TYPE Cnv_Errors_DUT :
STRUCT
	Error_Word_1:	UINT;
	Error_Word_2:	UINT;
	Error_Word_3:	UINT;
	Error_Word_4:	UINT;
END_STRUCT
END_TYPE

(* stored: Version 1.1.0.1
   DUT Cnv_Errors_DUT: Id {4c0f0708-8af3-4fdf-adc5-509ce8c61434} *)
